(* Logix 5000 project; controller Sine_wave_basic 1756-L85E rev 33.11; software revision 33.01 *)

TASK MainTask (continuous, watchdog 500 ms) : MainProgram

MODULES
   Local : 1756-L85E (ICP 4, rev 33.11)
END_MODULES

VAR_GLOBAL   (* controller tags *)
   frequency : REAL := 1.0;
   function : REAL := 60.769375;
   IoT_data : DINT := 61;
   time_index : REAL := 336.91702;
END_VAR

PROGRAM MainProgram   (* main routine MainRoutine *)
VAR
   sample_time : TIMER := (PRE := 100, ACC := 100, EN := 1, DN := 1);
END_VAR

ROUTINE MainRoutine   (* ladder *)
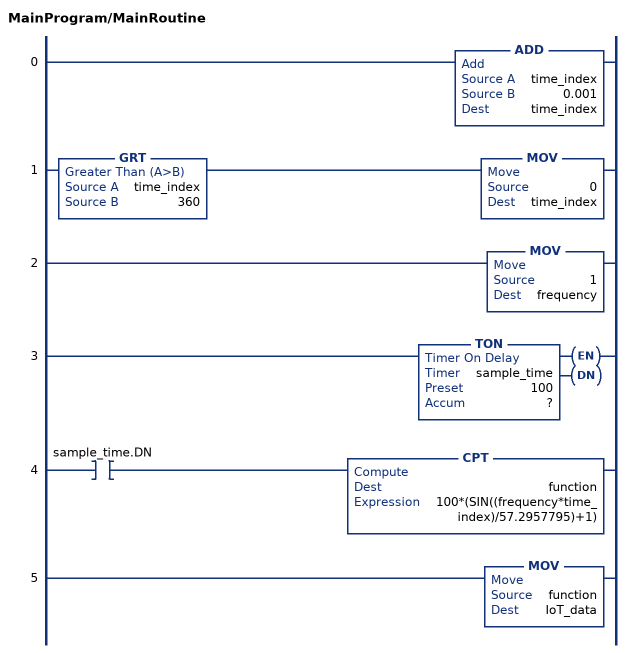
   0: ADD(time_index,0.001,time_index);
   1: GRT(time_index,360)MOV(0,time_index);
   2: MOV(1,frequency);
   3: TON(sample_time,?,?);
   4: XIC(sample_time.DN)CPT(function,100*(SIN((frequency*time_index)/57.2957795)+1));
   5: MOV(function,IoT_data);
END_ROUTINE
END_PROGRAM
